PROGRAM PRG_AdsClientTests
VAR
END_VAR

GVL_AdsClientTests.IsRunning := TRUE;

END_PROGRAM

(* stored: Version 1.1.0.1, ProductVersion 3.1.4024.9
   POU PRG_AdsClientTests: Id {d3e9ca6d-84a0-4f3a-9bdc-c7b060ad3f7f}, SpecialFunc None *)
